Staubli VAL3: SettingENC.pjx

--- SettingENC.pjx ---
Parameters version=s7.6 stackSize=5000 millimeterUnit=true
Program file=getErrorMessage.pgx
Program file=init.pgx
Program file=listFilling.pgx
Program file=readMe.pgx
Program file=start.pgx
Program file=stop.pgx
Data file=SettingENC.dtx
Library alias=ut path=Disk://Tracking/Tools/util/util.pjx

--- README.pgx ---
program readMe()
begin
  // Possible value for the variable sTxtBoxType
  // A : Alphanumerical value
  // N : Numerical value
  // B : Boolean
  // L : List
  // D : Display only (cannot be edited)
  // The coordinate (variable sTxtBoxPos) of the items are relative to the upper left corner
end
